// TIA Portal project "Projeto 2 - mistura" (V11)

(* hardware
DEVICE "ET 200S station_1"  ET200S-Station
   slot 0: "Rack"  Rail
   slot 2: "PLC_1"  IM151-8 F-CPU  6ES7 151-8FB01-0AB0  V3.2
      slot 1: "PROFINET interface_1"  PN-IO
         slot 1: "Port_1"  Port
         slot 2: "Port_2"  Port
         slot 3: "Port_3"  Port
   slot 4: "PM-E DC24V /8A RO_1"  6ES7 138-4CA80-0AB0
   slot 5: "4DI x 24VDC HF_1"  4DI DC24V HF  6ES7 131-4BD01-0AB0
   slot 6: "4DI x 24VDC HF_2"  4DI DC24V HF  6ES7 131-4BD01-0AB0
   slot 7: "4DI x 24VDC HF_3"  4DI DC24V HF  6ES7 131-4BD01-0AB0
   slot 8: "4DI x 24VDC HF_4"  4DI DC24V HF  6ES7 131-4BD01-0AB0
   slot 9: "4DI x 24VDC HF_5"  4DI DC24V HF  6ES7 131-4BD01-0AB0
   slot 10: "4DO x 24VDC / 0.5A HF_1"  4DO DC24V/0.5A HF  6ES7 132-4BD00-0AB0
   slot 11: "4DO x 24VDC / 0.5A HF_2"  4DO DC24V/0.5A HF  6ES7 132-4BD00-0AB0
   slot 12: "PM-E DC24V /8A RO_2"  6ES7 138-4CA80-0AB0
   slot 13: "4DO x 24VDC / 0.5A HF_3"  4DO DC24V/0.5A HF  6ES7 132-4BD00-0AB0
   slot 14: "4DO x 24VDC / 0.5A HF_4"  4DO DC24V/0.5A HF  6ES7 132-4BD00-0AB0
   slot 15: "4DO x 24VDC / 0.5A HF_5"  4DO DC24V/0.5A HF  6ES7 132-4BD00-0AB0
   slot 16: "2AI x U HF_1"  2AI U HF  6ES7 134-4LB02-0AB0
   slot 17: "2AI x U HF_2"  2AI U HF  6ES7 134-4LB02-0AB0
   slot 18: "2AO x U HF_1"  2AO U HF  6ES7 135-4LB02-0AB0
   slot 19: "1 Count 24V_1"  1 COUNT 24V/100 kHz C/F/M/W  6ES7 138-4DA04-0AB0  V2.0
   slot 20: "4SI IO link_1"  4SI IO-Link  6ES7 138-4GA50-0AB0
*)

// ===== PLC "PLC_1"  IM151-8 F-CPU =====

VAR_GLOBAL   // PLC tag table "Default tag table"
   "sa" AT %I1.0 : Bool;
   "sb" AT %I1.1 : Bool;
   "ph0" AT %I1.2 : Bool;
   "e1" AT %M0.1 : Bool;
   "e0" AT %M0.0 : Bool;
   "e2" AT %M0.2 : Bool;
   "ph1" AT %I1.3 : Bool;
   "e3" AT %M0.3 : Bool;
   "v1" AT %Q6.0 : Bool;
   "v2" AT %Q6.1 : Bool;
   "start" AT %I2.0 : Bool;
   "v3" AT %Q6.2 : Bool;
   "v4" AT %Q6.3 : Bool;
   "m" AT %Q7.0 : Bool;
   "e4" AT %M0.4 : Bool;
   "e5" AT %M0.5 : Bool;
   "e6" AT %M0.6 : Bool;
   "teste1" AT %M0.7 : Bool;
   "teste2" AT %M1.0 : Bool;
   "saida1" AT %Q7.1 : Bool;
   "saida2" AT %Q7.2 : Bool;
   "teste3" AT %M1.1 : Bool;
END_VAR

ORGANIZATION_BLOCK "Main"   // OB1, LAD
TITLE = "Main Program Sweep (Cycle)"
{ S7_Optimized_Access := 'FALSE' }
VERSION : 0.1
   VAR_TEMP
      OB1_EV_CLASS : Byte;   // Bits 0-3 = 1 (Coming event), Bits 4-7 = 1 (Event class 1)
      OB1_SCAN_1 : Byte;   // 1 (Cold restart scan 1 of OB 1), 3 (Scan 2-n of OB 1)
      OB1_PRIORITY : Byte;   // Priority of OB Execution
      OB1_OB_NUMBR : Byte;   // 1 (Organization block 1, OB1)
      OB1_RESERVED_1 : Byte;   // Reserved for system
      OB1_RESERVED_2 : Byte;   // Reserved for system
      OB1_PREV_CYCLE : Int;   // Cycle time of previous OB1 scan (milliseconds)
      OB1_MIN_CYCLE : Int;   // Minimum cycle time of OB1 (milliseconds)
      OB1_MAX_CYCLE : Int;   // Maximum cycle time of OB1 (milliseconds)
      OB1_DATE_TIME : Date_And_Time;   // Date and time OB1 started
   END_VAR
BEGIN
END_ORGANIZATION_BLOCK